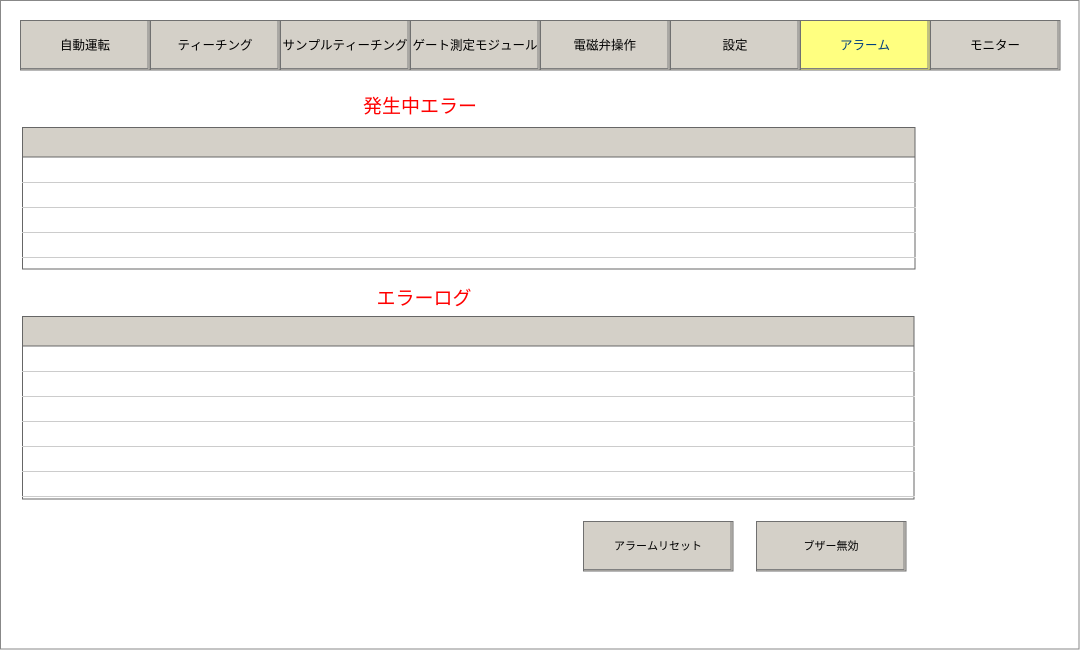
VISUALIZATION s_alarm  // 1080x650
    Rectangle (0,0 1080x650)
    Table (22,316 892x183), data array: gvl_error.var_ary_alarmlistLog
        p3854506369: gvl_error.var_ary_alarmlistLog[INDEX].var_alarmLevel
        p1892666644: gvl_error.var_ary_alarmlistLog[INDEX].var_alarmName
        p511219082: アラーム名
        p338671338: gvl_error.var_ary_alarmlistLog[INDEX].var_alarmMassge
        p2170511999: gvl_error.var_ary_alarmlistLog[INDEX].var_alarmTime
        p3723444502: gvl_error.var_ary_alarmlistLog[INDEX].var_alarmCode1
        p1218418051: gvl_error.var_ary_alarmlistLog[INDEX].var_alarmCode2
        p1755163831: 詳細
        p4092479075: 発生時刻
        p2237128397: 識別コード
        p505689113: エラーID
    Table (22,127 893x142), data array: gvl_error.var_ary_alarmlistActive
        p3854506369: gvl_error.var_ary_alarmlistActive[INDEX].var_alarmLevel
        p1892666644: gvl_error.var_ary_alarmlistActive[INDEX].var_alarmName
        p338671338: gvl_error.var_ary_alarmlistActive[INDEX].var_alarmMassge
        p2170511999: gvl_error.var_ary_alarmlistActive[INDEX].var_alarmTime
        p3723444502: gvl_error.var_ary_alarmlistActive[INDEX].var_alarmCode1
        p1218418051: gvl_error.var_ary_alarmlistActive[INDEX].var_alarmCode2
        p511219082: アラーム名
        p1755163831: 詳細
        p4092479075: 発生時刻
        p2237128397: 識別コード
        p505689113: エラーID
    Button (583,521 150x50), "アラームリセット"
        tap gvl_error.flg_reset
    Label (299,283 250x30), "エラーログ"
    Label (295,91 250x30), "発生中エラー"
    Button (20,20 130x50), "自動運転"
        OnMouseClick: change screen: s_auto
    Button (150,20 130x50), "ティーチング"
        OnMouseClick: change screen: s_teaching1
    Button (670,20 130x50), "設定"
        OnMouseClick: change screen: s_setting
    Button (540,20 130x50), "電磁弁操作"
        OnMouseClick: change screen: s_manual
    Button (410,20 130x50), "ゲート測定モジュール"
        OnMouseClick: change screen: s_gm_teaching
    Button (800,20 130x50), "アラーム", colour toggle: gvl_io.flg_signalTowerRed
        OnMouseClick: change screen: s_alarm
    Button (280,20 130x50), "サンプルティーチング"
        OnMouseClick: change screen: s_sample
    Button (756,521 150x50), "ブザー無効", colour toggle: gvl_visu.flg_btn_invalidBuzzer
        toggle gvl_visu.flg_btn_invalidBuzzer
    Button (930,20 130x50), "モニター"
        OnMouseClick: change screen: s_monitor
END_VISUALIZATION

(* stored: Version 1.1.0.1, ProductVersion 3.1.4024.11
   Visu s_alarm: Id {4124158c-eb85-4acf-8305-5319f0112d0e} *)
